{attribute 'qualified_only'}
{attribute 'strict'}
TYPE State :
(
	Error := 0,
	ManualMode,
	SetupMode,
	ProductionMode,
	ModusSelection
);
END_TYPE

(* stored: Version 1.1.0.1
   DUT State: Id {2932a2f4-44f3-4a70-9de3-0fdd595f4508} *)
